{attribute addProperty BoxType "EL3058-0000-0017"}
{attribute addProperty Id "AI_Standard_ChannelAT %I*ARRAY[0..7] OF AI_Standard_Channel_B51B79FC648810WcStateAT %I*WcState_98A4DF7520.250InfoDataAT %I*InfoData_BC63D37F80100"}
{attribute addProperty CRC "1498765698"}
{attribute addProperty SizeInBites "730"}
{attribute addProperty SizeInBytes "91.25"}
TYPE EL3058_6F92BA30 :
STRUCT
	{attribute addProperty Name "AI_Standard_Channel"}
	AI_Standard_Channel : ARRAY[0..7] OF AI_Standard_Channel_B51B79FC;
	{attribute addProperty Name "WcState"}
	WcState : WcState_98A4DF75;
	{attribute addProperty Name "InfoData"}
	InfoData : InfoData_BC63D37F;
END_STRUCT
END_TYPE

(* stored: Version 1.2.0.0, ProductVersion 3.1.4024.9
   DUT EL3058_6F92BA30: Id {75a27fea-727b-4dd7-995f-c3eb1b5bff54} *)
